% RSLogix 500 project PROJECT 1  CGT Part 1.RSS, saved by version 8.30.00.16 %
PROJECT "UNTITLED"    % processor: Bul.1763 MicroLogix 1100 Series B %

PROGRAM FILES
  LAD 2 "MAIN"  4 rungs
  LAD 3 "INPUT"  3 rungs
  LAD 4 "OUTPUTS"  3 rungs
  LAD 6 "LOGIC"  11 rungs

DATA FILES
  O0 OUTPUT  4 elements
  I1 INPUT  6 elements
  S2 STATUS  66 elements
  B3 BINARY  2 elements
  T4 TIMER  4 elements
  C5 COUNTER  1 elements
  R6 CONTROL  1 elements
  N7 INTEGER  1 elements
  F8 FLOAT  1 elements

LADDER 2 "MAIN"
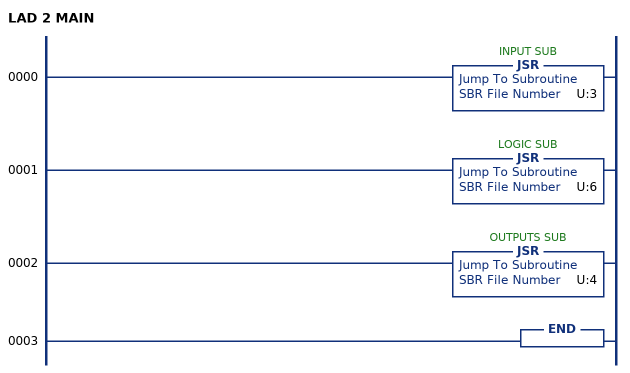
% Rung: 0 %
SOR JSR U:3 EOR
%   U:3  "INPUT SUB" %
% Rung: 1 %
SOR JSR U:6 EOR
%   U:6  "LOGIC SUB" %
% Rung: 2 %
SOR JSR U:4 EOR
%   U:4  "OUTPUTS SUB" %
% Rung: 3 %
SOR END EOR

LADDER 3 "INPUT"
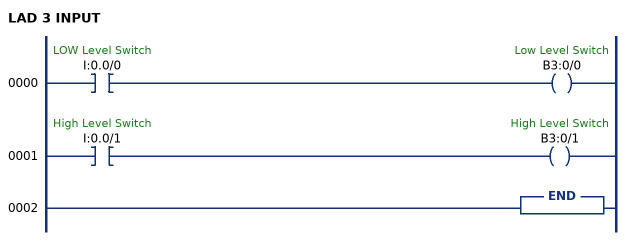
% Rung: 0 %
SOR XIC I:0.0/0 OTE B3:0/0 EOR
%   I:0.0/0  "LOW Level Switch" %
%   B3:0/0  "Low Level Switch" %
% Rung: 1 %
SOR XIC I:0.0/1 OTE B3:0/1 EOR
%   I:0.0/1  "High Level Switch" %
%   B3:0/1  "High Level Switch" %
% Rung: 2 %
SOR END EOR

LADDER 4 "OUTPUTS"
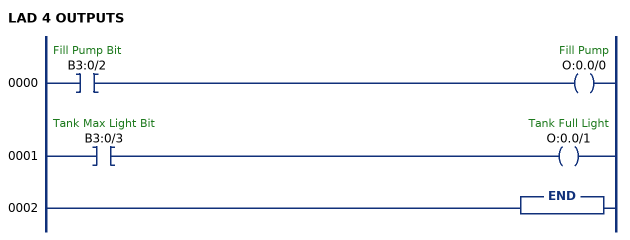
% Rung: 0 %
SOR XIC B3:0/2 OTE O:0.0/0 EOR
%   B3:0/2  "Fill Pump Bit" %
%   O:0.0/0  "Fill Pump" %
% Rung: 1 %
SOR XIC B3:0/3 OTE O:0.0/1 EOR
%   B3:0/3  "Tank Max Light Bit" %
%   O:0.0/1  "Tank Full Light" %
% Rung: 2 %
SOR END EOR

LADDER 6 "LOGIC"
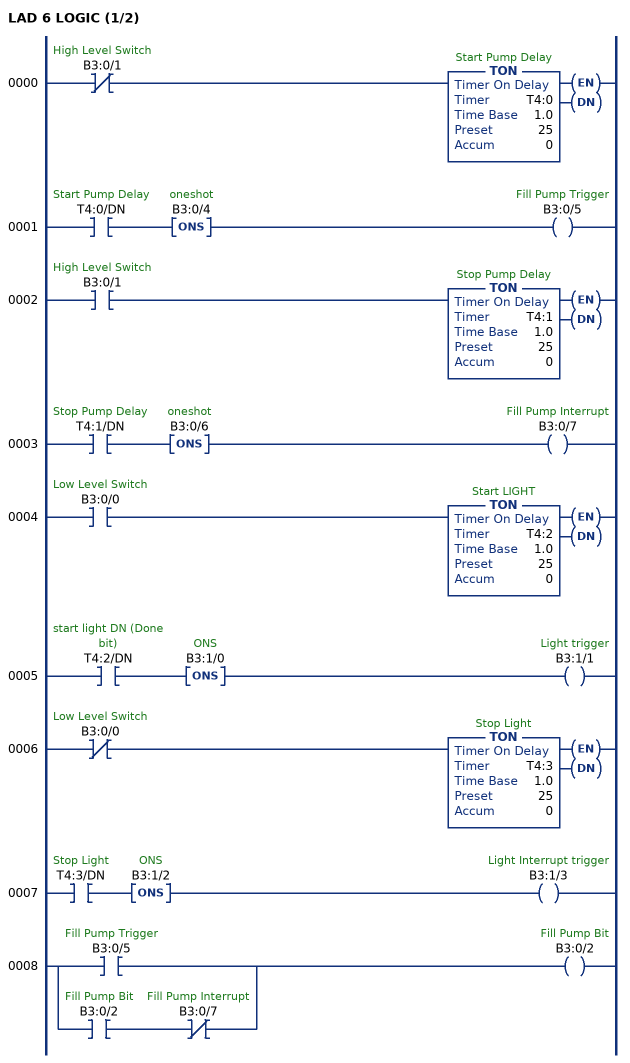
% Rung: 0 %
SOR XIO B3:0/1 TON T4:0 1.0 25 0 EOR
%   B3:0/1  "High Level Switch" %
%   T4:0  "Start Pump Delay" %
% Rung: 1 %
SOR XIC T4:0/DN ONS B3:0/4 OTE B3:0/5 EOR
%   T4:0  "Start Pump Delay" %
%   B3:0/4  "oneshot" %
%   B3:0/5  "Fill Pump Trigger" %
% Rung: 2 %
SOR XIC B3:0/1 TON T4:1 1.0 25 0 EOR
%   B3:0/1  "High Level Switch" %
%   T4:1  "Stop Pump Delay" %
% Rung: 3 %
SOR XIC T4:1/DN ONS B3:0/6 OTE B3:0/7 EOR
%   T4:1/DN  "Stop Pump Delay" %
%   B3:0/6  "oneshot" %
%   B3:0/7  "Fill Pump Interrupt" %
% Rung: 4 %
SOR XIC B3:0/0 TON T4:2 1.0 25 0 EOR
%   B3:0/0  "Low Level Switch" %
%   T4:2  "Start LIGHT" %
% Rung: 5 %
SOR XIC T4:2/DN ONS B3:1/0 OTE B3:1/1 EOR
%   T4:2/DN  "start light DN (Done bit)" %
%   B3:1/0  "ONS" %
%   B3:1/1  "Light trigger" %
% Rung: 6 %
SOR XIO B3:0/0 TON T4:3 1.0 25 0 EOR
%   B3:0/0  "Low Level Switch" %
%   T4:3  "Stop Light" %
% Rung: 7 %
SOR XIC T4:3/DN ONS B3:1/2 OTE B3:1/3 EOR
%   T4:3/DN  "Stop Light" %
%   B3:1/2  "ONS" %
%   B3:1/3  "Light Interrupt trigger" %
% Rung: 8 %
SOR BST XIC B3:0/5 NXB XIC B3:0/2 XIO B3:0/7 BND OTE B3:0/2 EOR
%   B3:0/5  "Fill Pump Trigger" %
%   B3:0/2  "Fill Pump Bit" %
%   B3:0/7  "Fill Pump Interrupt" %

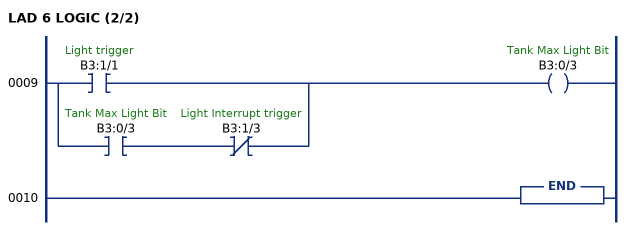
% Rung: 9 %
SOR BST XIC B3:1/1 NXB XIC B3:0/3 XIO B3:1/3 BND OTE B3:0/3 EOR
%   B3:1/1  "Light trigger" %
%   B3:0/3  "Tank Max Light Bit" %
%   B3:1/3  "Light Interrupt trigger" %
% Rung: 10 %
SOR END EOR

OTHER DOCUMENTED ADDRESSES
  T4:0/0  "pump start delay"

DATA TABLE (non-zero values as saved)
DATA B3
% B3:0 % 0X0040 0X0000
DATA T4
% .PRE .ACC %
% T4:0 % 25 0
% T4:1 % 25 0
% T4:2 % 25 0
% T4:3 % 25 0
